(* PLC project P1AM Function Blocks, OpenPLC P1AM Function Blocks Library 1.0, author Thiago Alves *)
(* stored: creationDateTime 2021-11-11T02:33:11, modificationDateTime 2021-11-11T02:33:11 *)

(* Initialize P1AM Modules and return the number of initialized modules on SUCCESS. If SUCCESS is zero, an error has occurred, or there aren't any modules on the bus *)
FUNCTION_BLOCK P1AM_INIT
  VAR_INPUT
    INIT : BOOL;
  END_VAR
  VAR_OUTPUT
    SUCCESS : SINT;
  END_VAR

            SUCCESS := 0;
          
END_FUNCTION_BLOCK

(* Get all inputs and update all outputs from P1-16CDR module. Also works with P1-15CDD1 and P1-15CDD2 *)
FUNCTION_BLOCK P1_16CDR
  VAR_INPUT
    SLOT : SINT;
    O1 : BOOL;
    O2 : BOOL;
    O3 : BOOL;
    O4 : BOOL;
    O5 : BOOL;
    O6 : BOOL;
    O7 : BOOL;
    O8 : BOOL;
  END_VAR
  VAR_OUTPUT
    I1 : BOOL;
    I2 : BOOL;
    I3 : BOOL;
    I4 : BOOL;
    I5 : BOOL;
    I6 : BOOL;
    I7 : BOOL;
    I8 : BOOL;
  END_VAR

            I1 := 0;
          
END_FUNCTION_BLOCK

(* Get all inputs from P1-08Nxx modules. Compatible with P1-08NA, P1-08ND3, P1-08NE3 and P1-08SIM *)
FUNCTION_BLOCK P1_08N
  VAR_INPUT
    SLOT : SINT;
  END_VAR
  VAR_OUTPUT
    I1 : BOOL;
    I2 : BOOL;
    I3 : BOOL;
    I4 : BOOL;
    I5 : BOOL;
    I6 : BOOL;
    I7 : BOOL;
    I8 : BOOL;
  END_VAR

            I1 := 0;
          
END_FUNCTION_BLOCK

(* Get all inputs from P1-16Nxx modules. Compatible with P1-16ND3 and P1-16NE3 *)
FUNCTION_BLOCK P1_16N
  VAR_INPUT
    SLOT : SINT;
  END_VAR
  VAR_OUTPUT
    I1 : BOOL;
    I2 : BOOL;
    I3 : BOOL;
    I4 : BOOL;
    I5 : BOOL;
    I6 : BOOL;
    I7 : BOOL;
    I8 : BOOL;
    I9 : BOOL;
    I10 : BOOL;
    I11 : BOOL;
    I12 : BOOL;
    I13 : BOOL;
    I14 : BOOL;
    I15 : BOOL;
    I16 : BOOL;
  END_VAR

            I1 := 0;
          
END_FUNCTION_BLOCK

(* Set all outputs on P1-08Txx modules. Compatible with P1-08TA, P1-08TD1, P1-08TD2 and P1-08TRS *)
FUNCTION_BLOCK P1_08TMZ
  VAR_INPUT
    SLOT : SINT;
    O1 : BOOL;
    O2 : BOOL;
    O3 : BOOL;
    O4 : BOOL;
    O5 : BOOL;
    O6 : BOOL;
    O7 : BOOL;
    O8 : BOOL;
  END_VAR
  VAR
    DUMMY : SINT;
  END_VAR

            DUMMY := SLOT;
          
END_FUNCTION_BLOCK

(* Set all outputs on P1-16TR modules. Also compatible with P1-15TD1 and P1-15TD2 *)
FUNCTION_BLOCK P1_16TR
  VAR_INPUT
    SLOT : SINT;
    O1 : BOOL;
    O2 : BOOL;
    O3 : BOOL;
    O4 : BOOL;
    O5 : BOOL;
    O6 : BOOL;
    O7 : BOOL;
    O8 : BOOL;
    O9 : BOOL;
    O10 : BOOL;
    O11 : BOOL;
    O12 : BOOL;
    O13 : BOOL;
    O14 : BOOL;
    O15 : BOOL;
    O16 : BOOL;
  END_VAR
  VAR
    DUMMY : SINT;
  END_VAR

            DUMMY := SLOT;
          
END_FUNCTION_BLOCK

(* Get all analog inputs from P1-04ADxx modules. Compatible with P1-04AD, P1-04ADL-1 and P1-04ADL-2 *)
FUNCTION_BLOCK P1_04AD
  VAR_INPUT
    SLOT : SINT;
  END_VAR
  VAR_OUTPUT
    I1 : UINT;
    I2 : UINT;
    I3 : UINT;
    I4 : UINT;
  END_VAR
  VAR
    DUMMY : SINT;
  END_VAR

            DUMMY := SLOT;
          
END_FUNCTION_BLOCK
